(* PLC project WS11, CODESYS CODESYS V3.5 SP16 Patch 6 *)
(* stored: creationDateTime 2025-01-31T08:51:34.1198928, version 1.2.0, modificationDateTime 2025-01-31T08:51:09.87209, organization TTControl S.r.l. *)

TYPE t_Power :
STRUCT
	// structure for POWER outputs
	Set			: lib500_types.IO_POWER_STATUS := (state := lib500_types.IO_POWER_STATE.IO_POWER_OFF);		// set power output state
	Get			: lib500_types.IO_POWER_STATUS := (state := lib500_types.IO_POWER_STATE.IO_POWER_OFF);		// get power output state 
	Feedback	: lib500_types.IO_ADC_STATUS;																// get power output voltage feetback
END_STRUCT
END_TYPE

TYPE t_PWM :
STRUCT
	// structure for PWM outputs
	DutyCycle		: WORD := 0;								// pin duty cycle
	Error			: lib500_types.IO_ERRORTYPE;				// pin errorcode
	CurrMeasurement	: lib500_types.IO_PWM_CURRENT_QUEUE_E;		// pin current measurement
	CurrentValue	: WORD;										// usable current value
	PWMFeedback		: lib500_types.IO_PWM_FEEDBACK;				// voltage feedback
END_STRUCT
END_TYPE

(*****************************************************************************************
*  Copyright (C) 2022 TTControl S.r.l. All rights reserved.
*  Julius Durst Str. 66, I-39042 Brixen/Bressanone (BZ), Italy, https://ttcontrol.4me.com/
*
*  PRE: 			none
*  POST: 			none
*  GLOBAL:			gPowerStage, gSensorSupply, gSafetySwitch0, gPotRed, gLedRed, gCan1
*  LIBRARIES:		none
*  DESCRIPTION: 	This POU inizializes the powerstage and configures an analog input
*                   in voltage mode and an output in PWM mode. It reads CAN ID 0x200
*                   and set the PWM output depending on Byte 0 / 1 of this CAN message.
*                   It writes the value of analog input (Byte 0 / 1) with CAN ID 0x100. 					
*  REVISION HISTORY:	
*  2015-05-11		TLE 	Creation.
*  2016-04-05		TLE		Update to target 1.0.0.0
*  2017-02-06		TLE		Update to target 1.2.0.0
*  2017-11-27		TLE		Update to target 1.3.0.0
*  2017-04-09		ADC		Update to target 1.4.0.0
*  2019-07-23		EPI		Update to target 1.6.1.0
*  2020-11-09		EPI		Update to target 1.7.1.0
*  2022-02-21		EPI		Add diagnostic state and pin errorcodes
*  2022-07-13		EPI		Update to target 1.8.0.0
*
*****************************************************************************************)
PROGRAM PLC_PRG
VAR
	InitPLC       : BOOL := TRUE;		(* Initialization variable *)
	fbCanTxId100  : CanTx;              (* Function block to send one CAN message *)
	fbCanTxId110  : CanTx;       (* Function block to send one CAN message *)
	fbCanTxId120  : CanTx;       (* Function block to send one CAN message *)
	fbCanTxId130  : CanTx;       (* Function block to send one CAN message *)
	TxData        : ARRAY[0..7] OF BYTE;(* Data to be transmitted *)
	TxData_ID_110        : ARRAY[0..7] OF BYTE;(* Data to be transmitted *)
	TxData_ID_120_echo        : ARRAY[0..7] OF BYTE;(* Data to be transmitted *)
	TxData_ID_130_echo        : ARRAY[0..7] OF BYTE;(* Data to be transmitted *)
	fbCanRxId200  : CanRx;              (* Function block to get one CAN message*)
	
END_VAR

                    GVL.gDiagState.diag_state;																// update variable and display show diag state

IF (initPLC = TRUE) THEN
	GVL.gPowerStage.Set.state    	:= lib500_types.IO_POWER_STATE.IO_POWER_ON;	    	// Switching on Power Stage
    GVL.gSafetySwitch0.Set.state 	:= lib500_types.IO_POWER_STATE.IO_POWER_ON;      	// Switching on Safety Switch for PWM use
	GVL.gSensorSupply.Set.state 	:= lib500_types.IO_POWER_STATE.IO_POWER_ON;       	// Switching on Sensor Supply
// use variables and show values
	// Power outputs
	GVL.gPowerStage.Set.error;															// Power Stage set error
	GVL.gPowerStage.Get.state;															// Power Stage get state
	GVL.gPowerStage.Feedback.value;														// Power Stage voltage feedback
	GVL.gSafetySwitch0.Set.error;														// Safety Switch set error
	GVL.gSafetySwitch0.Get.state;														// Safety Switch get state
	GVL.gSafetySwitch0.Feedback.value;													// Safety Switch voltage feedback
	GVL.gSensorSupply.Set.error;														// Sensor Supply set error
	GVL.gSensorSupply.Get.state;														// Sensor Supply get state
	GVL.gSensorSupply.Feedback.value;													// Sensor Supply voltage feedback
	// application IOs
	GVL.gPotRed.error;																	// Pot Red pin error
	GVL.gLedRed.Error;																	// Led Red pin error
	GVL.gLedRed.CurrMeasurement.error;													// Led Red current measurement error
	GVL.gLedRed.CurrMeasurement.values[0];												// Led Red current
	GVL.gLedRed.PWMFeedback.high_time;													// Led Red PWM feedback
	
// Initialize CAN 1	
	CanInit(	iEnable			:= TRUE,                                				// Initialiaze CAN 
				iChannel		:= 1, 													// CAN Channel 1
				iCAN			:= ADR(GVL.gCan1), 										// Structure for sending / receiving CAN messages
				iBaudrate       := 500, 												// 250 kBit
				iCanIdExtended  := FALSE, 												// Standard CAN Frame
				iEcuCycleTime   := T#10MS);												// Cycle time of task calling TX and RX
    InitPLC := FALSE;																	// Execute this block one time for initialisation
END_IF                                                                  				
                                                                        				
cl_split_word(	input	:= DWORD_TO_WORD(GVL.gPotRed.value),							// Split PotRed value in two bytes to send them over CAN
				byte0	=> TxData[0],                                   				
				byte1	=> TxData[1]);                                  				
				                                                        				
fbCanTxId100(	iEnable				:= TRUE, 											// Enables sending of messages
				iCAN				:= ADR(GVL.gCan1),									// Structure for sending / receiving CAN messages
				iForceSend			:= FALSE,                           				// Force sending sends message immediately
				iTransmitRate		:= T#100MS, 										// Cyclic transmission every 100ms
				iCanId				:= 16#100,											// CAN Id for message to send
				iCanIdExtended		:= FALSE, 											// Standard CAN Frame
				iByteCount			:= 8,												// Number of bytes to send
				iData				:= TxData, 											// Data frame
				oTransmitterId		=> ,                                				
				oTooManyTransmitters=> ,                                				
				oMsgSent			=> );        
				
				TxData_ID_110[0] := 15;
				TxData_ID_110[1] := 14;
				TxData_ID_110[2] := 13;
				TxData_ID_110[3] := 12;
				TxData_ID_110[4] := 11;
				TxData_ID_110[5] := 10;
				TxData_ID_110[6] := 9;
				TxData_ID_110[7] := 8;
				
fbCanTxId110(	iEnable				:= TRUE, 											// Enables sending of messages
				iCAN				:= ADR(GVL.gCan1),									// Structure for sending / receiving CAN messages
				iForceSend			:= FALSE,                           				// Force sending sends message immediately
				iTransmitRate		:= T#100MS, 										// Cyclic transmission every 100ms
				iCanId				:= 16#110,											// CAN Id for message to send
				iCanIdExtended		:= FALSE, 											// Standard CAN Frame
				iByteCount			:= 8,												// Number of bytes to send
				iData				:= TxData_ID_110, 									// Data frame
				oTransmitterId		=> ,                                				
				oTooManyTransmitters=> ,                                				
				oMsgSent			=> );                 

fbCanTxId120(	iEnable				:= TRUE, 											// Enables sending of messages
				iCAN				:= ADR(GVL.gCan1),									// Structure for sending / receiving CAN messages
				iForceSend			:= FALSE,                           				// Force sending sends message immediately
				iTransmitRate		:= T#100MS, 										// Cyclic transmission every 100ms
				iCanId				:= 16#130,											// CAN Id for message to send
				iCanIdExtended		:= FALSE, 											// Standard CAN Frame
				iByteCount			:= 8,												// Number of bytes to send
				iData				:= TxData_ID_130_echo, 									// Data frame
				oTransmitterId		=> ,                                				
				oTooManyTransmitters=> ,                                				
				oMsgSent			=> );                  

fbCanTxId130(	iEnable				:= TRUE, 											// Enables sending of messages
				iCAN				:= ADR(GVL.gCan1),									// Structure for sending / receiving CAN messages
				iForceSend			:= FALSE,                           				// Force sending sends message immediately
				iTransmitRate		:= T#100MS, 										// Cyclic transmission every 100ms
				iCanId				:= 16#120,											// CAN Id for message to send
				iCanIdExtended		:= FALSE, 											// Standard CAN Frame
				iByteCount			:= 8,												// Number of bytes to send
				iData				:= TxData_ID_120_echo, 									// Data frame
				oTransmitterId		=> ,                                				
				oTooManyTransmitters=> ,                                				
				oMsgSent			=> );                          				        				
				                                                        				
fbCanRxId200(	iCAN				:= ADR(GVL.gCan1),  								// Structure for sending / receiving CAN messages
				iCanId				:= 16#200,											// CAN Id of receiving message 
				iCanIdExtended		:= FALSE,  											// Standard CAN Frame
				iTimeoutLimit		:= T#500MS,											// Timeout after 500ms - Flag will be set 
				oByteCount			=> ,                                	
				oData				=> ,                                	
				oNewData			=> ,                                	
				oCanTimeout			=> ,                                	
				oReceiverId			=> ,                                	
				oTooManyReceivers	=> );	                            	
                                                                        	
IF fbCanRxId200.oNewData THEN															// If new CAN data is available
	GVL.gLedRed.DutyCycle := cl_make_word(	byte0 := fbCanRxId200.oData[0], 			// Make word using two over CAN received bytes and set it as LedRed setpoint*)
											byte1 := fbCanRxId200.oData[1]);					
	TxData_ID_120_echo := fbCanRxId200.oData;
	TxData_ID_130_echo := fbCanRxId200.oData;
	
ELSIF fbCanRxId200.oCanTimeout THEN														// If timeout flag is enabled switch off LedRed
	GVL.gLedRed.DutyCycle := 0;
END_IF
                  
END_PROGRAM

PROGRAM _ErrorCB_PRG
VAR
	diag_state : lib500_types.DIAG_STATETYPE := lib500_types.DIAG_STATETYPE.DIAG_STATE_DISABLED;
	watchdog_state : lib500_types.DIAG_WD_STATETYPE := lib500_types.DIAG_WD_STATETYPE.DIAG_WD_STATE_UNKNOWN;
	error : lib500_types.DIAG_ERRORCODE := (error_code := lib500_types.DIAG_ERRORTYPE.DIAG_E_NOERROR, 
                                            device_num := lib500_types.DIAG_DEVICETYPE.DIAG_DEV_NONE,
                                            faulty_value := 0);
	return_code : lib500_types.IO_ERRORTYPE := lib500_types.IO_ERRORTYPE.IO_E_UNKNOWN;
	
	reaction : lib500_types.DIAG_REACTION := lib500_types.DIAG_REACTION.DIAG_ERR_SAFESTATE;
	
	call_count : UDINT := 0;
END_VAR

                    (* get the reason for the error callback *)
return_code := lib500.DIAG_CDS_GetErrorReason(ADR(diag_state), 
                                              ADR(watchdog_state),
                                              ADR(error));

(* custom handler code can be placed here *)

(* the choices for the reactions are:
   -> lib500_types.DIAG_REACTION.DIAG_ERR_NOACTION
   -> lib500_types.DIAG_REACTION.DIAG_ERR_SAFESTATE
   -> lib500_types.DIAG_REACTION.DIAG_ERR_DISABLE_SSW0
   -> lib500_types.DIAG_REACTION.DIAG_ERR_DISABLE_SSW1
   -> lib500_types.DIAG_REACTION.DIAG_ERR_DISABLE_SSW2
   -> lib500_types.DIAG_REACTION.DIAG_ERR_DISABLE_HS00
   -> lib500_types.DIAG_REACTION.DIAG_ERR_DISABLE_HS01
   -> lib500_types.DIAG_REACTION.DIAG_ERR_DISABLE_HS02
   -> lib500_types.DIAG_REACTION.DIAG_ERR_DISABLE_HS03
   -> lib500_types.DIAG_REACTION.DIAG_ERR_DISABLE_HS04
   -> lib500_types.DIAG_REACTION.DIAG_ERR_DISABLE_HS05
   -> lib500_types.DIAG_REACTION.DIAG_ERR_DISABLE_HS06
   -> lib500_types.DIAG_REACTION.DIAG_ERR_DISABLE_HS07
   
   it's also possible to combine (binary-or) reactions, like:
   -> lib500_types.DIAG_REACTION.DIAG_ERR_DISABLE_SSW0 OR 
      lib500_types.DIAG_REACTION.DIAG_ERR_DISABLE_SSW1
*)

(* pass the error reaction to the DIAG system *)
lib500.DIAG_CDS_SetErrorReaction(reaction);

(* increment call count *)
call_count := call_count + 1;
                  
END_PROGRAM

PROGRAM _NotificationCB_PRG
VAR
	diag_state : lib500_types.DIAG_STATETYPE := lib500_types.DIAG_STATETYPE.DIAG_STATE_DISABLED;
	watchdog_state : lib500_types.DIAG_WD_STATETYPE := lib500_types.DIAG_WD_STATETYPE.DIAG_WD_STATE_UNKNOWN;
	error : lib500_types.DIAG_ERRORCODE := (error_code := lib500_types.DIAG_ERRORTYPE.DIAG_E_NOERROR, 
                                            device_num := lib500_types.DIAG_DEVICETYPE.DIAG_DEV_NONE,
                                            faulty_value := 0);
	return_code : lib500_types.IO_ERRORTYPE := lib500_types.IO_ERRORTYPE.IO_E_UNKNOWN;
	
	call_count : UDINT := 0;
END_VAR

                    (* get the reason for the notification callback *)
return_code := lib500.DIAG_CDS_GetNotificationReason(ADR(diag_state), 
                                                     ADR(watchdog_state),
                                                     ADR(error));

(* custom handler code can be placed here *)

(* increment call count *)
call_count := call_count + 1;
                  
END_PROGRAM

(*****************************************************************************************
*  Copyright (C) 2022 TTControl S.r.l. All rights reserved.
*  Julius Durst Str. 66, I-39042 Brixen/Bressanone (BZ), Italy, https://ttcontrol.4me.com/
*
*  PRE: 			none
*  POST: 			none
*  GLOBAL:			none
*  LIBRARIES:		none
*  DESCRIPTION: 	This POU describes the use of this workshop example.
*					
*  REVISION HISTORY:	
*  2015-05-11		TLE 	Creation.
*  2016-04-05		TLE		Update to target 1.0.0.0
*  2017-02-06		TLE		Update to target 1.2.0.0
*  2017-11-27		TLE		Update to target 1.3.0.0
*  2017-04-09		ADC		Update to target 1.4.0.0
*  2019-07-23		EPI		Update to target 1.6.1.0
*  2020-11-09		EPI		Update to target 1.7.1.0
*  2022-02-21		EPI		Add diagnostic state and pin errorcodes
*  2022-07-13		EPI		Update to target 1.8.0.0
*
*****************************************************************************************)
PROGRAM ReadMe

                    (* * * * * * * * * * * * * * * * * * * * * * * * * * * * * * * * * * * * * * * * * * 
 *	READ ME			READ ME			READ ME			READ ME			READ ME               
 * * * * * * * * * * * * * * * * * * * * * * * * * * * * * * * * * * * * * * * * * * 
 * 
 *  This program shows how to read and write CAN 2.0b messages. It uses Pin 103
 *  as voltage mode input and Pin 153 as PWM output.
 *	
 * * * * * * * * * * * * * * * * * * * * * * * * * * * * * * * * * * * * * * * * * * )
                  
END_PROGRAM

(*****************************************************************************************
*  Copyright (C) 2022 TTControl S.r.l. All rights reserved.
*  Julius Durst Str. 66, I-39042 Brixen/Bressanone (BZ), Italy, https://ttcontrol.4me.com/
*
*  PRE: 			none
*  POST: 			none
*  GLOBAL:			none
*  LIBRARIES:		none
*  DESCRIPTION: 	Disclaimer
*					
*  REVISION HISTORY:	
*  2017-01-31		TLE 	Creation.
*
*****************************************************************************************)

PROGRAM Disclaimer
VAR
END_VAR

                    (* * * * * * * * * * * * * * * * * * * * * * * * * * * * * * * * * * * * * * * * * * 
 *	DISCLAIMER		DISCLAIMER		DISCLAIMER		DISCLAIMER  	DISCLAIMER       
 * * * * * * * * * * * * * * * * * * * * * * * * * * * * * * * * * * * * * * * * * *  
 
This document is proprietary to TTControl GmbH and no ownership rights are hereby transferred.
No part of this document shall be used, reproduced, translated, converted, adapted, stored in an
information storage or a retrieval system, communicated or transmitted in any form or by any means
(electronic or mechanical, including photocopying, recording), for any commercial purpose, including
without limitation, sale, resale, license, rental or lease, without the prior express written consent
of TTControl GmbH.

TTControl GmbH does not make any representations, warranties or guarantees, express or implied,
as to the accuracy or completeness of the document. The information in this document is subject to
change without notice and does not represent a commitment on the part of TTControl GmbH. Users
must be aware that updates and amendments will be made from time to time to the document. It is
the user’s responsibility to determine whether there have been any such updates or amendments.
Neither TTControl GmbH nor any of its directors, officers, employees or agents shall be liable in
contract, tort or in any other manner whatsoever to any person for any loss, damage, injury, liability,
cost or expense of any nature, including without limitation incidental, special, direct or consequential
damages arising out of or in connection with the use of this document.


Der Inhalt dieses Dokuments ist geistiges Eigentum der TTControl GmbH und es werden hieran keine Eigentumsrechte 
übertragen. Dieses Dokument, einschließlich seiner Teile, darf in keiner Form und auf keine Weise (elektronisch 
oder mechanisch, einschließlich Fotokopien und Aufnahmen) füR kommerzielle Zwecke  verwendet, vervielfältigt, 
übersetzt, verändert oder adaptiert werden. "Kommerzielle Zwecke" umfassen insbesondere Verkauf, Weiterverkauf, 
Lizenz, Miete oder Pacht ohne die vorherige ausdrückliche schriftliche Zustimmung von TTControl GmbH. Es ist nicht 
erlaubt dieses Dokument, einschließlich seiner Teile, in einem Datenspeicher oder einem Datenabfragesystem zu 
speichern, es zu übertragen oder zu versenden. 

TTControl GmbH übernimmt, soweit gesetzlich zulässig, weder ausdrücklich noch stillschweigend Gewährleistungen 
oder Garantien betreffend die Richtigkeit oder Vollständigkeit des Dokuments. Die TTControl behäLT sich das Recht 
vor, ohne Benachrichtigung den Inhalt des Dokuments abzuändern, ohne dass ihr hieraus irgendwelche Verpflichtungen 
erwachsen. Der Benutzer muss sich bewusst sein, dass Aktualisierungen und Anpassungen gelegentlich erfolgen werden. 
Es obliegt dem Benutzer festzustellen, ob solche Aktualisierungen oder Anpassungen erfolgt sind. Soweit gesetzlich 
zulässig, haftet weder die TTControl GmbH noch einer ihrer Geschäftsführer, Angestellten  oder Repräsentanten vertraglich, 
schadenersatzrechtlich oder auf irgendeiner anderen Grundlage füR Verluste, Schäden,  Kosten oder Ausgaben jeglicher Art, 
einschließlich, aber nicht beschränkt auf Neben-, Folge- oder Sonderschäden, direkte oder indirekte Schäden, die aus oder 
im Zusammenhang mit diesem Dokument entstehen.

 * * * * * * * * * * * * * * * * * * * * * * * * * * * * * * * * * * * * * * * * * * 
 *	DISCLAIMER		DISCLAIMER		DISCLAIMER		DISCLAIMER  	DISCLAIMER               
 * * * * * * * * * * * * * * * * * * * * * * * * * * * * * * * * * * * * * * * * * *)
                  
END_PROGRAM

CONFIGURATION Device
  RESOURCE Application ON PLC
(* global variable list GVL *)
VAR_GLOBAL
	gDiagState 			: lib500_types.DIAG_STATUS;			// ECU diagnostic status
                                                            	
    gPowerStage     	: t_Power;							// Powerstage status structure
	gSafetySwitch0  	: t_Power;							// Safety Switch 0 status structure
    gSensorSupply       : t_Power;   						// Sensor Supply status structure
    gPotRed        		: lib500_types.IO_ADC_STATUS;       // Red Potentiometer value
    gLedRed        		: t_PWM;	                        // Led Red output
	gCan1          		: tCan;                             // Structure for sending / receiving CAN messages
END_VAR
(* global variable list CONSTANTS *)
{attribute 'qualified_only'}
VAR_GLOBAL CONSTANT
	MAJOR : BYTE := 1;			// SW Version major
	MINOR : BYTE := 0;			// SW Version minor
	PATCH : BYTE := 8;			// SW Version patch
END_VAR
    TASK MainTask(INTERVAL := T#10ms, PRIORITY := 2);
    TASK _ErrorCallback(PRIORITY := 1);
    TASK _NotificationCallback(PRIORITY := 0);
    PROGRAM PLC_PRG WITH MainTask : PLC_PRG;
    PROGRAM _ErrorCB_PRG WITH _ErrorCallback : _ErrorCB_PRG;
    PROGRAM _NotificationCB_PRG WITH _NotificationCallback : _NotificationCB_PRG;
  END_RESOURCE
END_CONFIGURATION

CONFIGURATION CANs
END_CONFIGURATION

CONFIGURATION CAN0
END_CONFIGURATION

CONFIGURATION CAN1
END_CONFIGURATION

CONFIGURATION CAN2
END_CONFIGURATION

CONFIGURATION CAN3
END_CONFIGURATION

CONFIGURATION CAN4
END_CONFIGURATION

CONFIGURATION CAN5
END_CONFIGURATION

CONFIGURATION CAN6
END_CONFIGURATION

CONFIGURATION System
END_CONFIGURATION

CONFIGURATION Analog_Inputs_2Mode_10V
END_CONFIGURATION

CONFIGURATION Pin 107
END_CONFIGURATION

CONFIGURATION PotRed
END_CONFIGURATION

CONFIGURATION Pin 131
END_CONFIGURATION

CONFIGURATION <Empty>
END_CONFIGURATION

CONFIGURATION Pin 108
END_CONFIGURATION

CONFIGURATION <Empty>
END_CONFIGURATION

CONFIGURATION Pin 132
END_CONFIGURATION

CONFIGURATION <Empty>
END_CONFIGURATION

CONFIGURATION Pin 109
END_CONFIGURATION

CONFIGURATION <Empty>
END_CONFIGURATION

CONFIGURATION Pin 133
END_CONFIGURATION

CONFIGURATION <Empty>
END_CONFIGURATION

CONFIGURATION Pin 110
END_CONFIGURATION

CONFIGURATION <Empty>
END_CONFIGURATION

CONFIGURATION Pin 134
END_CONFIGURATION

CONFIGURATION <Empty>
END_CONFIGURATION

CONFIGURATION Analog_Inputs_2Mode_32V
END_CONFIGURATION

CONFIGURATION Pin 111
END_CONFIGURATION

CONFIGURATION <Empty>
END_CONFIGURATION

CONFIGURATION Pin 135
END_CONFIGURATION

CONFIGURATION <Empty>
END_CONFIGURATION

CONFIGURATION Pin 112
END_CONFIGURATION

CONFIGURATION <Empty>
END_CONFIGURATION

CONFIGURATION Pin 136
END_CONFIGURATION

CONFIGURATION <Empty>
END_CONFIGURATION

CONFIGURATION Pin 113
END_CONFIGURATION

CONFIGURATION <Empty>
END_CONFIGURATION

CONFIGURATION Pin 137
END_CONFIGURATION

CONFIGURATION <Empty>
END_CONFIGURATION

CONFIGURATION Pin 114
END_CONFIGURATION

CONFIGURATION <Empty>
END_CONFIGURATION

CONFIGURATION Pin 138
END_CONFIGURATION

CONFIGURATION <Empty>
END_CONFIGURATION

CONFIGURATION Analog_Inputs_3Mode
END_CONFIGURATION

CONFIGURATION Pin 103
END_CONFIGURATION

CONFIGURATION <Empty>
END_CONFIGURATION

CONFIGURATION Pin 127
END_CONFIGURATION

CONFIGURATION <Empty>
END_CONFIGURATION

CONFIGURATION Pin 104
END_CONFIGURATION

CONFIGURATION <Empty>
END_CONFIGURATION

CONFIGURATION Pin 128
END_CONFIGURATION

CONFIGURATION <Empty>
END_CONFIGURATION

CONFIGURATION Pin 105
END_CONFIGURATION

CONFIGURATION <Empty>
END_CONFIGURATION

CONFIGURATION Pin 129
END_CONFIGURATION

CONFIGURATION <Empty>
END_CONFIGURATION

CONFIGURATION Pin 106
END_CONFIGURATION

CONFIGURATION <Empty>
END_CONFIGURATION

CONFIGURATION Pin 130
END_CONFIGURATION

CONFIGURATION <Empty>
END_CONFIGURATION

CONFIGURATION Digital_Outputs_HS
END_CONFIGURATION

CONFIGURATION Pin 149
END_CONFIGURATION

CONFIGURATION <Empty>
END_CONFIGURATION

CONFIGURATION Pin 173
END_CONFIGURATION

CONFIGURATION <Empty>
END_CONFIGURATION

CONFIGURATION Pin 152
END_CONFIGURATION

CONFIGURATION <Empty>
END_CONFIGURATION

CONFIGURATION Pin 176
END_CONFIGURATION

CONFIGURATION <Empty>
END_CONFIGURATION

CONFIGURATION Pin 155
END_CONFIGURATION

CONFIGURATION <Empty>
END_CONFIGURATION

CONFIGURATION Pin 179
END_CONFIGURATION

CONFIGURATION <Empty>
END_CONFIGURATION

CONFIGURATION Pin 158
END_CONFIGURATION

CONFIGURATION <Empty>
END_CONFIGURATION

CONFIGURATION Pin 182
END_CONFIGURATION

CONFIGURATION <Empty>
END_CONFIGURATION

CONFIGURATION Digital_Outputs_LS
END_CONFIGURATION

CONFIGURATION Pin 251
END_CONFIGURATION

CONFIGURATION <Empty>
END_CONFIGURATION

CONFIGURATION Pin 238
END_CONFIGURATION

CONFIGURATION <Empty>
END_CONFIGURATION

CONFIGURATION Pin 252
END_CONFIGURATION

CONFIGURATION <Empty>
END_CONFIGURATION

CONFIGURATION Pin 239
END_CONFIGURATION

CONFIGURATION <Empty>
END_CONFIGURATION

CONFIGURATION Pin 253
END_CONFIGURATION

CONFIGURATION <Empty>
END_CONFIGURATION

CONFIGURATION Pin 240
END_CONFIGURATION

CONFIGURATION <Empty>
END_CONFIGURATION

CONFIGURATION Pin 254
END_CONFIGURATION

CONFIGURATION <Empty>
END_CONFIGURATION

CONFIGURATION Pin 241
END_CONFIGURATION

CONFIGURATION <Empty>
END_CONFIGURATION

CONFIGURATION PVG_Outputs
END_CONFIGURATION

CONFIGURATION Pin 161
END_CONFIGURATION

CONFIGURATION <Empty>
END_CONFIGURATION

CONFIGURATION Pin 185
END_CONFIGURATION

CONFIGURATION <Empty>
END_CONFIGURATION

CONFIGURATION Pin 188
END_CONFIGURATION

CONFIGURATION <Empty>
END_CONFIGURATION

CONFIGURATION Pin 164
END_CONFIGURATION

CONFIGURATION <Empty>
END_CONFIGURATION

CONFIGURATION Pin 191
END_CONFIGURATION

CONFIGURATION <Empty>
END_CONFIGURATION

CONFIGURATION Pin 167
END_CONFIGURATION

CONFIGURATION <Empty>
END_CONFIGURATION

CONFIGURATION Pin 194
END_CONFIGURATION

CONFIGURATION <Empty>
END_CONFIGURATION

CONFIGURATION Pin 170
END_CONFIGURATION

CONFIGURATION <Empty>
END_CONFIGURATION

CONFIGURATION PWM_Outputs
END_CONFIGURATION

CONFIGURATION Safety_switch_0
END_CONFIGURATION

CONFIGURATION Pin 153
END_CONFIGURATION

CONFIGURATION LedRed
END_CONFIGURATION

CONFIGURATION Pin 177
END_CONFIGURATION

CONFIGURATION <Empty>
END_CONFIGURATION

CONFIGURATION Pin 156
END_CONFIGURATION

CONFIGURATION <Empty>
END_CONFIGURATION

CONFIGURATION Pin 180
END_CONFIGURATION

CONFIGURATION <Empty>
END_CONFIGURATION

CONFIGURATION Pin 159
END_CONFIGURATION

CONFIGURATION <Empty>
END_CONFIGURATION

CONFIGURATION Pin 183
END_CONFIGURATION

CONFIGURATION <Empty>
END_CONFIGURATION

CONFIGURATION Pin 186
END_CONFIGURATION

CONFIGURATION <Empty>
END_CONFIGURATION

CONFIGURATION Pin 162
END_CONFIGURATION

CONFIGURATION <Empty>
END_CONFIGURATION

CONFIGURATION Pin 189
END_CONFIGURATION

CONFIGURATION <Empty>
END_CONFIGURATION

CONFIGURATION Pin 165
END_CONFIGURATION

CONFIGURATION <Empty>
END_CONFIGURATION

CONFIGURATION Pin 192
END_CONFIGURATION

CONFIGURATION <Empty>
END_CONFIGURATION

CONFIGURATION Pin 168
END_CONFIGURATION

CONFIGURATION <Empty>
END_CONFIGURATION

CONFIGURATION Pin 195
END_CONFIGURATION

CONFIGURATION <Empty>
END_CONFIGURATION

CONFIGURATION Pin 171
END_CONFIGURATION

CONFIGURATION <Empty>
END_CONFIGURATION

CONFIGURATION Safety_switch_1
END_CONFIGURATION

CONFIGURATION Pin 154
END_CONFIGURATION

CONFIGURATION <Empty>
END_CONFIGURATION

CONFIGURATION Pin 178
END_CONFIGURATION

CONFIGURATION <Empty>
END_CONFIGURATION

CONFIGURATION Pin 157
END_CONFIGURATION

CONFIGURATION <Empty>
END_CONFIGURATION

CONFIGURATION Pin 181
END_CONFIGURATION

CONFIGURATION <Empty>
END_CONFIGURATION

CONFIGURATION Pin 160
END_CONFIGURATION

CONFIGURATION <Empty>
END_CONFIGURATION

CONFIGURATION Pin 184
END_CONFIGURATION

CONFIGURATION <Empty>
END_CONFIGURATION

CONFIGURATION Pin 187
END_CONFIGURATION

CONFIGURATION <Empty>
END_CONFIGURATION

CONFIGURATION Pin 163
END_CONFIGURATION

CONFIGURATION <Empty>
END_CONFIGURATION

CONFIGURATION Pin 190
END_CONFIGURATION

CONFIGURATION <Empty>
END_CONFIGURATION

CONFIGURATION Pin 166
END_CONFIGURATION

CONFIGURATION <Empty>
END_CONFIGURATION

CONFIGURATION Pin 193
END_CONFIGURATION

CONFIGURATION <Empty>
END_CONFIGURATION

CONFIGURATION Pin 169
END_CONFIGURATION

CONFIGURATION <Empty>
END_CONFIGURATION

CONFIGURATION Pin 196
END_CONFIGURATION

CONFIGURATION <Empty>
END_CONFIGURATION

CONFIGURATION Pin 172
END_CONFIGURATION

CONFIGURATION <Empty>
END_CONFIGURATION

CONFIGURATION Safety_switch_2
END_CONFIGURATION

CONFIGURATION Pin 101
END_CONFIGURATION

CONFIGURATION <Empty>
END_CONFIGURATION

CONFIGURATION Pin 125
END_CONFIGURATION

CONFIGURATION <Empty>
END_CONFIGURATION

CONFIGURATION Pin 150
END_CONFIGURATION

CONFIGURATION <Empty>
END_CONFIGURATION

CONFIGURATION Pin 174
END_CONFIGURATION

CONFIGURATION <Empty>
END_CONFIGURATION

CONFIGURATION Pin 102
END_CONFIGURATION

CONFIGURATION <Empty>
END_CONFIGURATION

CONFIGURATION Pin 126
END_CONFIGURATION

CONFIGURATION <Empty>
END_CONFIGURATION

CONFIGURATION Pin 151
END_CONFIGURATION

CONFIGURATION <Empty>
END_CONFIGURATION

CONFIGURATION Pin 175
END_CONFIGURATION

CONFIGURATION <Empty>
END_CONFIGURATION

CONFIGURATION Timer_Inputs_Cur
END_CONFIGURATION

CONFIGURATION Pin 115
END_CONFIGURATION

CONFIGURATION <Empty>
END_CONFIGURATION

CONFIGURATION Pin 139
END_CONFIGURATION

CONFIGURATION <Empty>
END_CONFIGURATION

CONFIGURATION Pin 116
END_CONFIGURATION

CONFIGURATION <Empty>
END_CONFIGURATION

CONFIGURATION Pin 140
END_CONFIGURATION

CONFIGURATION <Empty>
END_CONFIGURATION

CONFIGURATION Pin 117
END_CONFIGURATION

CONFIGURATION <Empty>
END_CONFIGURATION

CONFIGURATION Pin 141
END_CONFIGURATION

CONFIGURATION <Empty>
END_CONFIGURATION

CONFIGURATION Timer_Inputs
END_CONFIGURATION

CONFIGURATION Pin 122
END_CONFIGURATION

CONFIGURATION <Empty>
END_CONFIGURATION

CONFIGURATION Pin 146
END_CONFIGURATION

CONFIGURATION <Empty>
END_CONFIGURATION

CONFIGURATION Pin 123
END_CONFIGURATION

CONFIGURATION <Empty>
END_CONFIGURATION

CONFIGURATION Pin 147
END_CONFIGURATION

CONFIGURATION <Empty>
END_CONFIGURATION

CONFIGURATION Pin 124
END_CONFIGURATION

CONFIGURATION <Empty>
END_CONFIGURATION

CONFIGURATION Pin 148
END_CONFIGURATION

CONFIGURATION <Empty>
END_CONFIGURATION
